(* IEC 61131-3 sources: teller/JD_Teller_LC2_V11/Class/ChannelBaseData, 1 file *)

(* ---- ChannelBaseData.st ---- *)
(*!
<Class
	Name               = "ChannelBaseData"
	Revision           = "1.0"
	RealtimeTask       = "false"
	CyclicTask         = "false"
	BackgroundTask     = "false"
	Sigmatek           = "true"
	OSInterface        = "false"
	HighPriority       = "false"
	Automatic          = "false"
	UpdateMode         = "Prescan"
	IconPath           = ".\Class\Tool.ico"
	SharedCommandTable = "true"
	Objectsize         = "(284,120)">
	<Channels>
		<Server Name="Data" Visualized="false" Initialize="false" WriteProtected="true" Retentive="false"/>
	</Channels>
	<RevDoku>
		<Owner Company="Sigmatek" Author="BleErn"/>
		<Dokumentation Revision="1.0" Date="04.03.2010" Author="BleErn" Company="Sigmatek" Description="New Base Class for Input/Output-Channel-Classes"/>
	</RevDoku>
</Class>
*)
ChannelBaseData : CLASS
  //Servers:
	Data 	: SvrChCmd_DINT;
  //Clients:
  //Variables:
  //Functions:

	FUNCTION VIRTUAL GLOBAL Init;

	FUNCTION VIRTUAL GLOBAL UpdateCy
		VAR_INPUT
			Handle 	: DINT;
		END_VAR;

	FUNCTION VIRTUAL GLOBAL UpDateRt
		VAR_INPUT
			Handle 	: DINT;
		END_VAR;

	FUNCTION VIRTUAL GLOBAL UpDateRtPostScan
		VAR_INPUT
			handle 	: DINT;
		END_VAR;
  //Tables:
	FUNCTION @STD
		VAR_OUTPUT
			ret_code	: CONFSTATES;
		END_VAR;
	FUNCTION GLOBAL TAB @CT_;
END_CLASS;

FUNCTION VIRTUAL GLOBAL ChannelBaseData::Init

END_FUNCTION

#pragma warning(disable: 73 )
FUNCTION VIRTUAL GLOBAL ChannelBaseData::UpDateRt
	VAR_INPUT
		Handle 	: DINT;
	END_VAR

END_FUNCTION
#pragma warning(default: 73 )

#pragma warning(disable: 73 )
FUNCTION VIRTUAL GLOBAL ChannelBaseData::UpdateCy
	VAR_INPUT
		Handle 	: DINT;
	END_VAR

END_FUNCTION
#pragma warning(default: 73 )

#pragma warning(disable: 73 )
FUNCTION VIRTUAL GLOBAL ChannelBaseData::UpDateRtPostScan
	VAR_INPUT
		handle 	: DINT;
	END_VAR

END_FUNCTION
#pragma warning(default: 73 )
